FUNCTION_BLOCK FB_WeighingOversampling
VAR
	arrSamples AT %I* : ARRAY[1..OVERSAMPLING_FACTOR] OF DINT;
	arrBuffer : ARRAY[1..MAX_BUFFER_SIZE] OF REAL;
	rCycleAvg : LREAL;
	rAccumulate: LREAL;
	i	:INT;
	fbLoadFiler 		: FB_FilterEx;
	index :INT:=1;
	rRunningAcc	: LREAL;
	bFilled : BOOL;
	rRunningMeasure : LREAL;
	rRunningMeasureWithTare : LREAL;
	rTest:REAL;
	iCycles: UINT;
	iReqCycles :UINT;
	bGetMeasurement:BOOL;
	bMeasurementReady: BOOL;;
	rSingleMess: REAL;
	rSingleMessResult: REAL;
	fbRunningAnalog : fbAnalogMeasurement;
	fbSingleAnalog  : fbAnalogMeasurement;
	
	bReqMeasurement : BOOL;
	fbReqMeasurement :R_TRIG;

	fbTON_ForceSampling	: TON;
	fbTON_ForceStable	: TON;
	rLastRunningMeasure: REAL;
	bMeasurementError : BOOL;
	fbSingleMeasurementTimeout: TON;
	rZeroValueScalled:REAL;
END_VAR
VAR PERSISTENT
	stSettings:  ST_WeighingSettings;
	rZeroValue 		: REAL;
END_VAR
VAR CONSTANT
	OVERSAMPLING_FACTOR: INT:=1;
	MAX_BUFFER_SIZE:INT:=1000;
END_VAR


rAccumulate := 0;
FOR i := 1 TO OVERSAMPLING_FACTOR DO
    rAccumulate := rAccumulate + arrSamples[i];
END_FOR
rCycleAvg := rAccumulate/OVERSAMPLING_FACTOR ;

//Running Measurment
rRunningAcc := rRunningAcc - arrBuffer[index];
rRunningAcc := rRunningAcc + rCycleAvg;
arrBuffer[index] := rCycleAvg ;
index := index + 1;
IF index > MAX_BUFFER_SIZE THEN
	index :=1;
	bFilled := TRUE;
END_IF
IF bFilled THEN
	rRunningMeasure := rRunningAcc/MAX_BUFFER_SIZE;
END_IF

fbTON_ForceSampling(IN:= NOT fbTON_ForceSampling.Q, PT:= T#30MS);
IF fbTON_ForceSampling.Q THEN
	fbTON_ForceStable(IN:= ABS(rLastRunningMeasure-rRunningMeasure)< MAX(0.5,rRunningMeasure*0.005), PT:= INT_TO_TIME(stSettings.iWeightStabilisationTimeMS));
	rLastRunningMeasure := rRunningMeasure;
END_IF



//Single Measurment
fbSingleMeasurementTimeout(IN:=bGetMeasurement AND NOT prForceIsStable AND iCycles = 0,PT:= T#5S);

fbReqMeasurement(CLK:=bReqMeasurement);
IF fbReqMeasurement.Q THEN
	bGetMeasurement := TRUE;
	bMeasurementError := FALSE;
	bMeasurementReady := FALSE;
END_IF
IF bGetMeasurement AND prForceIsStable THEN
	rSingleMess := rSingleMess + rCycleAvg;
	iCycles := iCycles +1;
	IF iCycles >= iReqCycles THEN
		rSingleMessResult := rSingleMess/iCycles;
		bMeasurementReady := TRUE;
		bGetMeasurement:= FALSE;
		iCycles :=0;
		rSingleMess := 0.0;
	END_IF
ELSIF bGetMeasurement AND NOT prForceIsStable AND iCycles > 0 OR fbSingleMeasurementTimeout.Q THEN
	bMeasurementError := TRUE;
	bGetMeasurement:= FALSE;
	iCycles :=0;
	rSingleMess := 0.0;
END_IF

//Scalling
fbSingleAnalog(rIn:=rSingleMessResult-rZeroValue,stMeasureScalingData:=stSettings.stScalling, tStalaCzasowa:=T#1MS);
fbRunningAnalog(rIn:=rRunningMeasure-rZeroValue,stMeasureScalingData:=stSettings.stScalling, tStalaCzasowa:=T#1MS);
rZeroValueScalled := fScalling(rIn:=rZeroValue,stMeasureScalingData:=stSettings.stScalling);
//HMI
IF stSettings.bManualSingleMeasureRequest AND_THEN mGetMeasurement(1000) THEN
	stSettings.bManualSingleMeasureRequest:=FALSE;
END_IF
IF stSettings.bTareRequest AND_THEN mTare() THEN
	stSettings.bTareRequest:=FALSE;
END_IF

METHOD mGetMeasurement : BOOL
VAR_INPUT
	iCycles: INT;
END_VAR
VAR
	bInit:BOOL:=FALSE;
END_VAR

bReqMeasurement := TRUE;
iReqCycles := iCycles;
mGetMeasurement := FALSE;
IF bMeasurementReady OR bMeasurementError THEN
	mGetMeasurement := TRUE;
	bMeasurementReady := bReqMeasurement := FALSE;
END_IF;
END_METHOD

METHOD mTare : BOOL
VAR_INPUT
END_VAR
mTare:=FALSE;
IF mGetMeasurement(1000) THEN
	IF NOT prSingleMeasurementError THEN
		rZeroValue := prSingleMeasurementRaw;
	END_IF
	mTare:=TRUE;
END_IF
END_METHOD

PROPERTY prForceIsStable : BOOL
GET
prForceIsStable := fbTON_ForceStable.Q;
END_GET
END_PROPERTY

PROPERTY prRunningMeasurement : REAL
GET
prRunningMeasurement := fbRunningAnalog.rOutFiltered;
END_GET
END_PROPERTY

PROPERTY prSingleMeasurement : REAL
GET
prSingleMeasurement := fbSingleAnalog.rOutFiltered;
END_GET
END_PROPERTY

PROPERTY prSingleMeasurementError : BOOL
GET
prSingleMeasurementError := bMeasurementError;
END_GET
END_PROPERTY

PROPERTY prSingleMeasurementRaw : REAL
GET
prSingleMeasurementRaw := rSingleMessResult;
END_GET
END_PROPERTY

END_FUNCTION_BLOCK

(* stored: Version 1.1.0.1, ProductVersion 3.1.4024.15
   POU FB_WeighingOversampling: Id {3519dee1-614f-442c-be8a-15af5c35d0c3}, SpecialFunc None
   Method mGetMeasurement: Id {b755d138-d4ca-4b3a-9962-72c9a6f2bf0b}
   Method mTare: Id {9b6dea7e-18b9-466a-aba8-9e503c4931be}
   Property prForceIsStable: Id {6c1dbff3-59e6-4566-9180-c7daab8a55bf}
   Get Get: Id {4fb681c2-9cf1-4ee4-9515-20464fe7afda}
   Property prRunningMeasurement: Id {bcc25dcf-27df-4f0a-858c-49c915207399}
   Get Get: Id {1221aa39-6940-4645-9480-b2c10f3a9d64}
   Property prSingleMeasurement: Id {dfd4f5d1-d18d-4698-9a97-7bd6b9c12f74}
   Get Get: Id {253c9750-b34b-4117-8494-502b0d5e4059}
   Property prSingleMeasurementError: Id {be6856fd-b8eb-4733-9767-175d2464b50a}
   Get Get: Id {49bc2472-d6e4-4733-8e2d-f367c54a123c}
   Property prSingleMeasurementRaw: Id {56186388-389d-4ad3-a899-5843ef86ec71}
   Get Get: Id {f9136aac-b5d3-4c8f-98bc-6e528a51fe72} *)
